(* IEC 61131-3 sources: Eteam-Testing-Suite/, 4 files *)

(* ---- FB_TestLogger.st ---- *)
FUNCTION_BLOCK FB_TestLogger
VAR_INPUT
    StepDescription : STRING(80);  // Step label
    StepResult      : BOOL;        // TRUE = Pass, FALSE = Fail
    AddStep         : BOOL;        // Rising edge = Add to log
    WriteLogToFile  : BOOL;        // Rising edge = Save to file
    PrintToLogger   : BOOL;        // Rising edge = Print log to TwinCAT system
END_VAR

VAR_OUTPUT
    LogComplete     : BOOL;        // TRUE once writing is done
    StepCount       : INT;         // How many steps logged
    Busy            : BOOL;        // Writing file
    Error           : BOOL;        // File error occurred
END_VAR

VAR
    // Internal logging arrays
    LogStep   : ARRAY[0..99] OF STRING(80);
    LogValue  : ARRAY[0..99] OF BOOL;
    LogIndex  : INT := 0;

    // File handling
    fbOpen  : FB_FileOpen;
    fbWrite : FB_FileWrite;
    fbClose : FB_FileClose;
    hFile   : UINT;
    i       : INT;
    logStr  : STRING(255);
    writeState : INT := 0;

    // Edge detection
    lastAddStep       : BOOL := FALSE;
    lastWriteLog      : BOOL := FALSE;
    lastPrintToLogger : BOOL := FALSE;
END_VAR

// Detect rising edges
VAR
    risingAdd    : BOOL := AddStep AND NOT lastAddStep;
    risingWrite  : BOOL := WriteLogToFile AND NOT lastWriteLog;
    risingPrint  : BOOL := PrintToLogger AND NOT lastPrintToLogger;
END_VAR

lastAddStep := AddStep;
lastWriteLog := WriteLogToFile;
lastPrintToLogger := PrintToLogger;

LogComplete := FALSE;
Error := FALSE;
Busy := FALSE;
StepCount := LogIndex;

(* === Add Step to Log === *)
IF risingAdd AND (LogIndex < 100) THEN
    LogStep[LogIndex] := StepDescription;
    LogValue[LogIndex] := StepResult;
    LogIndex := LogIndex + 1;
END_IF

(* === Print to TwinCAT Logger === *)
IF risingPrint THEN
    FOR i := 0 TO LogIndex - 1 DO
        TcEventLog.Add(16#00000001, 'Step: ' + LogStep[i] + ' | Result: ' + BOOL_TO_STRING(LogValue[i]));
    END_FOR;
END_IF

(* === Write to CSV File === *)
CASE writeState OF
    0:
        IF risingWrite THEN
            fbOpen.sFileName := 'C:\TestLogs\TestLog.csv';
            fbOpen.ePath := PATH_GENERIC;
            fbOpen.eOpenMode := FOPEN_MODEAPPEND;
            fbOpen(bExecute := TRUE);
            writeState := 1;
        END_IF

    1:
        fbOpen(bExecute := FALSE);
        IF NOT fbOpen.bBusy THEN
            IF fbOpen.bError THEN
                Error := TRUE;
                writeState := 0;
            ELSE
                hFile := fbOpen.hFile;
                i := 0;
                writeState := 2;
            END_IF
        END_IF

    2:
        IF i < LogIndex THEN
            logStr := CONCAT(CONCAT(LogStep[i], ','), BOOL_TO_STRING(LogValue[i]));
            fbWrite.hFile := hFile;
            fbWrite.pBuffer := ADR(logStr);
            fbWrite.nBufferSize := LEN(logStr);
            fbWrite(bExecute := TRUE);
            writeState := 3;
        ELSE
            writeState := 5;
        END_IF

    3:
        fbWrite(bExecute := FALSE);
        IF NOT fbWrite.bBusy THEN
            IF fbWrite.bError THEN
                Error := TRUE;
                writeState := 5;
            ELSE
                i := i + 1;
                writeState := 2;
            END_IF
        END_IF

    5:
        fbClose.hFile := hFile;
        fbClose(bExecute := TRUE);
        writeState := 6;

    6:
        fbClose(bExecute := FALSE);
        IF NOT fbClose.bBusy THEN
            LogComplete := TRUE;
            writeState := 0;
        END_IF
END_CASE

(* ---- Section_1.st ---- *)
FUNCTION_BLOCK FB_Execute_Section_1
VAR_INPUT
    StartTest : BOOL;
    Input1    : BOOL; // Tie to mapped I/O variable (e.g., SF1)
    Input2    : BOOL; // Tie to mapped I/O variable (e.g., SF2)
    Input3    : BOOL;
    Input4    : BOOL;
END_VAR
VAR_OUTPUT
    Done      : BOOL;
    Result    : BOOL;
END_VAR

VAR
    state : INT := 0;
    timer : TON;
END_VAR

// Example logic with 10-second wait
timer(IN := (state = 1), PT := T#1s);

CASE state OF
    0: // Wait for start
        IF StartTest THEN
            Done := FALSE;
            Result := FALSE;
            state := 1;
        END_IF

    1: // Wait 1s
        timer();
        IF timer.Q THEN
            // Here you could check some I/O signals or conditions
            Result := Input1 AND Input2 AND Input3 AND Input4; // Example: test passed
            Done := TRUE;
            state := 2;
        END_IF

    2: // Hold until reset
        IF NOT StartTest THEN
            state := 0;
        END_IF
END_CASE

(* ---- Test Program.st ---- *)
VAR
    SF1: BOOL; (* Mine Phone Continuity SF1 (1008 (2) port 8) *)
    SF2: BOOL; (* Mine Phone Continuity SF2 (1008 (2) port 7) *)
    SF6: BOOL; (* MGT Continuity SF6 (1008 (3) port 1) *)
    SF8: BOOL; (* MGT Continuity SF8 (1008 (3) port 2) *)
    SF4: BOOL; (* Fire pull Station SF4 (1008 (1) port 1) *)
    SF5: BOOL; (* Fire Alarm Sound SF5 (2024 port 2) *)
    J1_1: BOOL; (* Lighting 24V Check J1 (1) (1008 (3) port 3) *)
    J1_2: BOOL; (* Lighting 24V Check J1 (2) (1008 (3) port 4) *)
    J2_1: BOOL; (* Lighting 24V Check J2 (1) (1008 (3) port 5) *)
    J2_2: BOOL; (* Lighting 24V Check J2 (2) (1008 (3) port 6) *)
    J3_1: BOOL; (* 24V PWR Check J3 (1) (1008 (1) port 4) *)
    J3_2: BOOL; (* 24V PWR Check J3 (2) (1008 (1) port 5) *)
    J4_1: BOOL; (* 24V PWR Check J4 (1) (1008 (1) port 6) *)
    J4_2: BOOL; (* 24V PWR Check J4 (2) (1008 (1) port 7) *)
    J5_1: BOOL; (* 24V PWR Check J5 (1) (1008 (2) port 1) *)
    J5_2: BOOL; (* 24V PWR Check J5 (2) (1008 (2) port 2) *)
    J6_1: BOOL; (* 24V PWR Check J6 (1) (1008 (2) port 3) *)
    J6_2: BOOL; (* 24V PWR Check J6 (2) (1008 (2) port 4) *)
    J7_4: BOOL; (* 24V PWR Check J7 (4) (1008 (1) port 2) *)
    J7_5: BOOL; (* 24V PWR Check J7 (5) (1008 (1) port 3) *)
    J8_4: BOOL; (* 24V PWR Check J8 (4) (1008 (2) port 5) *)
    J8_5: BOOL; (* 24V PWR Check J8 (5) (1008 (2) port 6) *)
    Door_Switch: BOOL; (* Door Switch, Unknown Port *)
    Estop_Signal: BOOL; (* Estop Signal, Unknown Port *)
    DCDC_Signal: BOOL; (* DCDC Signal, Unknown Port *)
    Estop_Signal_Low: BOOL; (* Estop Signal Low, Unknown Port *)
    DCDC_Signal_Low: BOOL; (* DCDC Signal Low, Unknown Port *)
    DCDC_Calibration_Manual: BOOL; (* DCDC Calibration Manual, Unknown Port *)
    DCDC_2_Signal: BOOL; (* DCDC 2 Signal, Unknown Port *)
    DCDC_2_Signal_Low: BOOL; (* DCDC 2 Signal Low, Unknown Port *)
    DCDC_2_Calibration_Manual: BOOL; (* DCDC 2 Calibration Manual, Unknown Port *)
    PSU_1_Signal: BOOL; (* PSU 1 Signal, Unknown Port *)
    PSU_1_Signal_Low: BOOL; (* PSU 1 Signal Low, Unknown Port *)
    PSU_2_Signal: BOOL; (* PSU 2 Signal, Unknown Port *)
    PSU_2_Signal_Low: BOOL; (* PSU 2 Signal Low, Unknown Port *)
    Hear_Fire_Alarm_Manual: BOOL; (* Hear Fire Alarm Manual, Unknown Port *)
    Ping_address_1: BOOL; (* Ping address 1, Unknown Port *)
    Ping_address_2: BOOL; (* Ping address 2, Unknown Port *)
    Ping_address_3: BOOL; (* Ping address 3, Unknown Port *)
    Ping_address_4: BOOL; (* Ping address 4, Unknown Port *)
    grace_port_visible: BOOL; (* grace port visible, Unknown Port *)
    120V_indicator_visible: BOOL; (* 120V indicator visible, Unknown Port *)
    programmed_psu1_manual: BOOL; (* programmed psu1 manual, Unknown Port *)
    programmed_psu2_manual: BOOL; (* programmed psu2 manual, Unknown Port *)
    24v_load_test_psu1: BOOL; (* 24v load test psu1, Unknown Port *)
    24v_load_test_psu2: BOOL; (* 24v load test psu2, Unknown Port *)
    ecat_branch_test: BOOL; (* ecat branch test, Unknown Port *)
    ecat_branch_test_2: BOOL; (* ecat branch test 2, Unknown Port *)
    mine_phone_battery_manual: BOOL; (* mine phone battery manual, Unknown Port *)
    ping_ips: BOOL; (* ping ips, Unknown Port *)
    gfci_test_manual: BOOL; (* gfci test manual, Unknown Port *)

    TestingStage   : INT := 0;
    StepReady      : BOOL := TRUE;
    AdvanceStep    : BOOL; // Could be a physical input or HMI button

    // Logging arrays
    LogStep        : ARRAY[0..39] OF STRING(50);
    LogValue       : ARRAY[0..39] OF BOOL;

    // Internal helpers
    LogIndex       : INT := 0;

    Section1 : FB_Execute_Section_1;
    TestInProgress : BOOL;

END_VAR

// Main program

// Variable	Purpose
// StartTest	External trigger to begin
// Done	Goes TRUE when test finishes
// Result	TRUE = pass, FALSE = fail
// state	Local step tracking inside FB
// TON	Timer used for delays

// Advance only on rising edge of AdvanceStep
IF AdvanceStep AND StepReady THEN
    CASE TestingStage OF

        0:
            Section1(StartTest := TRUE,
                     Input1 := SF1,
                     Input2 := SF2,
                     Input3 := SF6,
                     Input4 := SF8);

            IF Section1.Done THEN
                LogStep[LogIndex] := 'section 1'
                LogValue[LogIndex] := Section1.Result;
                LogIndex := LogIndex + 1;
                TestingStage := 1;
            END_IF;

        ELSE
            // End of test
            TestingStage := 0;
            LogIndex := 0;
            LogStep[LogIndex] := 'Test Complete';
            LogValue[LogIndex] := TRUE;
            LogIndex := LogIndex + 1;
            TestingStage := 0;
            //

        END_CASE;

        StepReady := FALSE; // Lock step until AdvanceStep is Released
    END_IF
    // Allow next step when button released
    IF NOT AdvanceStep THEN
        StepReady:= TRUE;
    END_IF

// This is where I call the test logger program to create the test log

// VAR
//     TestLogger : FB_TestLogger;
//     AdvanceStep : BOOL;
//     ManualTrigger : BOOL;
// END_VAR

// Call it like this:

// pascal
// Copy
// Edit
// // During test step
// IF AdvanceStep THEN
//     TestLogger.StepDescription := 'Power Input 1 good';
//     TestLogger.StepResult := TRUE;
//     TestLogger.AddStep := TRUE;
// ELSE
//     TestLogger.AddStep := FALSE;
// END_IF

// // Trigger saving the log
// TestLogger.WriteLogToFile := ManualTrigger;

// // Optionally print it to logger
// TestLogger.PrintToLogger := FALSE; // or TRUE on demand

// TestLogger();

(* ---- Test Saving Log.st ---- *)
VAR
    fbFileOpen  : FB_FileOpen;
    fbFileWrite : FB_FileWrite;
    fbFileClose : FB_FileClose;
    fileHandle  : UINT;

    filePath    : T_MaxString := 'C:\TestLogs\TestLog.csv'; // Ensure this folder exists
    writeDone   : BOOL := FALSE;
    logString   : STRING(255);
    i           : INT;
END_VAR

// Step 2: Open the File

fbFileOpen.sFileName := filePath;
fbFileOpen.ePath := PATH_GENERIC; // PATH_GENERIC = C:\ on your dev PC
fbFileOpen.eOpenMode := FOPEN_MODEAPPEND; // Append mode
fbFileOpen(bExecute := TRUE);
IF fbFileOpen.bBusy = FALSE AND fbFileOpen.bError = FALSE THEN
    fileHandle := fbFileOpen.hFile;
END_IF

// Step 3: Format & Write the Log Entries

FOR i := 0 TO LogIndex - 1 DO
    logString := CONCAT(CONCAT(LogStep[i], ','), BOOL_TO_STRING(LogValue[i]));
    fbFileWrite.hFile := fileHandle;
    fbFileWrite.pBuffer := ADR(logString);
    fbFileWrite.nBufferSize := LEN(logString);
    fbFileWrite(bExecute := TRUE);

    // Wait for write to finish before next iteration (simplified for cyclic task)
    IF fbFileWrite.bBusy = FALSE AND fbFileWrite.bError = FALSE THEN
        fbFileWrite(bExecute := FALSE); // reset
    END_IF
END_FOR

// Close the File
fbFileClose.hFile := fileHandle;
fbFileClose(bExecute := TRUE);
